{attribute 'Tc2GvlVarNames'}
VAR_GLOBAL
END_VAR

(* stored: Version 1.1.0.1, ProductVersion 3.1.4022.9
   GVL Global_Variables: Id {bb59e6e5-b6de-4c1a-a076-162eedc72354} *)
